# EPICS substitutions: TS02K-CS-IOC-01App/Db/TS02K-CS-IOC-01_expanded.substitutions
# This file was automatically generated on Thu 13 Aug 2026 12:19:05 BST from
# source: /dls_sw/prod/R3.14.12.7/support/IDLAB-BUILDER/1-77/etc/makeIocs/TS02K-CS-IOC-01.xml
#
# *** Please do not edit this file: edit the source file instead. ***
#

# Macros:
#  prefix  record prefix
file $(IDPLC)/db/idplc_axisEna.template
{
pattern { prefix }
    { "TS02K-MO-" }
}

# Macros:
#  prefix  pv prefix e.g. TS02K-MO-
file $(IDPLC)/db/idplc_status.template
{
pattern { prefix }
    { "TS02K-MO-" }
}

# Macros:
#  IOC  Device prefix
file $(IOCSTATS)/db/iocAdminSoft.db
{
pattern { IOC }
    { "TS02K-CS-IOC-01" }
}

# Macros:
#  IOC  Device prefix
file $(IOCSTATS)/db/iocAdminScanMon.db
{
pattern { IOC }
    { "TS02K-CS-IOC-01" }
}

# # Macros:
# #  name      name for gui elements
# #  EDM_FILE  edm screen, defaults to ioc_stats_softdls.edl
# #  IOC       ioc name
# file $(DEVIOCSTATS)/db/iocGui.db
# {
# pattern { name, EDM_FILE, IOC }
#     { "IOC.TS02K", "ioc_stats_softdls.edl", "TS02K-CS-IOC-01" }
# }

# Macros:
#  name    Name
#  port    Port Name
#  device  PV Prefix
file $(ETHER_IP)/db/ether_ip_plcInfo.template
{
pattern { name, port, device }
    { "PLC.INFO", "pport", "TS02K-MP-PLC-01" }
}

# Macros:
#  device  device prefix
#  port    port name of ether_ip driver
#  name    Object name and associated gui name
file $(DLSPLC)/db/NX102_controller_status.template
{
pattern { device, port, name }
    { "TS02K-MO-PLC-01:CS", "pport", "cont" }
}

# Macros:
#  device  Template argument
#  port    Template argument
#  tagidx  Template argument
#  name    Template argument
#  tag     Template argument
file $(DLSPLC)/db/NX102_digitalIn.template
{
pattern { device, port, tagidx, name, tag }
    { "TS02K-MO-PLC-01:ST1", "pport", "1", "CPMU6.S1", "Digital_In_Epics" }
    { "TS02K-MO-PLC-01:ST2", "pport", "2", "CPMU6.S2", "Digital_In_Epics" }
    { "TS02K-MO-PLC-01:ST3", "pport", "3", "CPMU6.S3", "Digital_In_Epics" }
}

# Macros:
#  device      device prefix
#  port        port name of ether_ip driver
#  interlock   Interlock suffix (e.g. :INT1)
#  tag         NX PLC tag string e.g. ILK (from ILK.Control[1])
#  tagidx      NX PLC tag index number e.g. 1 (from ILK.Control[1])
#  desc        Permit description (e.g. Front end permit)
#  name        Object name and gui association name
#  auto_reset  Set to 1 to push the reset button whenever the raw interlocks are all ok
file $(DLSPLC)/db/NX102_interlock.template
{
pattern { device, port, interlock, tag, tagidx, desc, name, auto_reset }
    { "TS02K-MO-PLC-01:MAIN", "pport", "", "ILK", "2", "Motion Interlocks", "CPMU6.0MOT", "0" }
    { "TS02K-MO-PLC-01:LIM", "pport", "", "ILK", "3", "Limit Interlocks", "CPMU6.1LIM", "0" }
    { "TS02K-MO-TILT-01", "pport", "", "ILK", "1", "Tilt Interlocks", "CPMU6.2TILT", "0" }
    { "TS02K-MO-PLC-01:SLIM", "pport", "", "ILK", "4", "Soft Limit Interlocks", "CPMU6.3SLIM", "0" }
}

# Macros:
#  prefix  Template argument
file $(IDPLC)/db/NX102_idoverrides.template
{
pattern { prefix }
    { "TS02K-MO" }
}

# Macros:
#  prefix  device prefix, e.g. SR02K-MO
#  port    port name of ether_ip driver
#  name    gui name
#  idname  id name
file $(IDPLC)/db/NX102_tilt.template
{
pattern { prefix, port, name, idname }
    { "TS02K-MO", "pport", "CPMU6.TILT", "CPMU6" }
}

# Macros:
#  prefix  Template argument
#  port    Template argument
file $(IDPLC)/db/NX102_axisexp.template
{
pattern { prefix, port }
    { "TS02K-MO", "pport" }
}

# Macros:
#  prefix  device prefix, e.g. SR02K-MO
#  port    port name of ether_ip driver
file $(IDPLC)/db/NX102_tiltpot.template
{
pattern { prefix, port }
    { "TS02K-MO", "pport" }
}

# Macros:
#  prefix  device prefix, e.g. SR02K-MO
#  port    port name of ether_ip driver
#  name    gui component name
#  idname  gui label
file $(IDPLC)/db/NX102_id.template
{
pattern { prefix, port, name, idname }
    { "TS02K-MO", "pport", "CPMU6.TAGS", "" }
}

# Macros:
#  prefix  device prefix, e.g. SR02K-MO
#  axx     axis, e.g. 1
#  port    port name of ether_ip driver
#  name    gui
file $(IDPLC)/db/NX102_idpotscan.template
{
pattern { prefix, axx, port, name }
    { "TS02K-MO", "1", "pport", "CPMU6.pot1" }
    { "TS02K-MO", "2", "pport", "CPMU6.pot2" }
    { "TS02K-MO", "3", "pport", "CPMU6.pot3" }
    { "TS02K-MO", "4", "pport", "CPMU6.pot4" }
}
